{attribute 'qualified_only'}
{attribute 'strict'}
TYPE E_ArmState :
(
	Idle			:= 0,
	FirstState		:= 1,
	Redo			:= 2,
	SecondState		:= 3,
	Done			:= 4,
	
	Reverse			:= 5,
	Inverse			:= 6
) := Idle;
END_TYPE

(* stored: Version 1.1.0.1, ProductVersion 3.1.4024.12
   DUT E_ArmState: Id {46dcca8c-b5a3-4d10-8c2c-84e0ab9c23ef} *)
